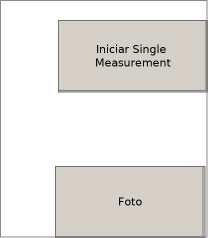
VISUALIZATION HMI  // 208x238
    Button (55,166 150x72), "Foto"
        tap MAIN.foto
    Button (58,20 150x72), "Iniciar Single Measurement"
        toggle MAIN.Single
END_VISUALIZATION

(* stored: Version 1.1.0.1, ProductVersion 3.1.4024.9
   Visu HMI: Id {9b423606-8548-47a2-b22c-955610dd6c90} *)
